{attribute addProperty BoxType "EL2595-0000-0019"}
{attribute addProperty Id "DOX_StatusAT %I*DOX_Status_95DEE7BC1620DOX_ControlAT %Q*DOX_Control_4111B8D51620WcStateAT %I*WcState_98A4DF7520.250InfoDataAT %I*InfoData_BC63D37F80100"}
{attribute addProperty CRC "2221615076"}
{attribute addProperty SizeInBites "114"}
{attribute addProperty SizeInBytes "14.25"}
TYPE EL2595_D45C87C7 :
STRUCT
	{attribute addProperty Name "DOX_Status"}
	DOX_Status : DOX_Status_95DEE7BC;
	{attribute addProperty Name "DOX_Control"}
	DOX_Control : DOX_Control_4111B8D5;
	{attribute addProperty Name "WcState"}
	WcState : WcState_98A4DF75;
	{attribute addProperty Name "InfoData"}
	InfoData : InfoData_BC63D37F;
END_STRUCT
END_TYPE

(* stored: Version 1.2.0.0, ProductVersion 3.1.4024.9
   DUT EL2595_D45C87C7: Id {2e0fe617-cc18-4488-af71-12a0e3078d2e} *)
